FUNCTION_BLOCK FB_Test
VAR_INPUT
END_VAR
VAR_OUTPUT
	iRes : INT;
END_VAR
VAR
		nMode : BYTE := 0;
		b0 : BIT;
		b1 : BIT;
		b2 : BIT;
	
END_VAR


nMode.0 := b0;
nMode.1 := b1;
nMode.2 := b2;

iRes := nMode;

END_FUNCTION_BLOCK

(* stored: Version 1.1.0.1, ProductVersion 3.1.4024.12
   POU FB_Test: Id {dae950d6-a500-4f8e-a352-072c6bc46b15}, SpecialFunc None *)
